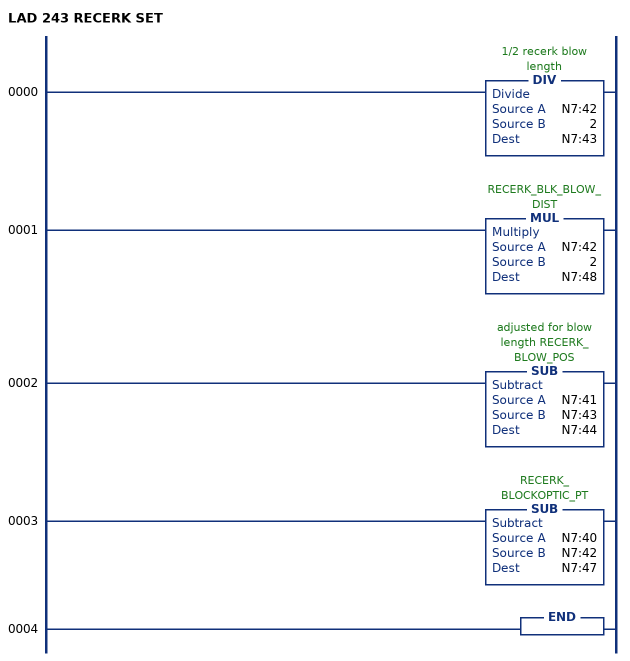
% Rung: 0 %
SOR DIV N7:42 2 N7:43 EOR
%   N7:42  RECERK_BLOW_LENGTH %
%   N7:43  "1/2 recerk blow length" %
% Rung: 1 %
SOR MUL N7:42 2 N7:48 EOR
%   N7:42  RECERK_BLOW_LENGTH %
%   N7:48  RECERK_BLK_BLOW_DIST %
% Rung: 2 %
SOR SUB N7:41 N7:43 N7:44 EOR
%   N7:41  RECERK_BLOW_POS_HMI  "recerk blow position set from hmi" %
%   N7:43  "1/2 recerk blow length" %
%   N7:44  RECERK_BLOW_POS  "adjusted for blow length" %
% Rung: 3 %
SOR SUB N7:40 N7:42 N7:47 EOR
%   N7:40  RECERK_OPTIC_POS %
%   N7:42  RECERK_BLOW_LENGTH %
%   N7:47  RECERK_BLOCKOPTIC_PT %
% Rung: 4 %
SOR END EOR

LADDER 244
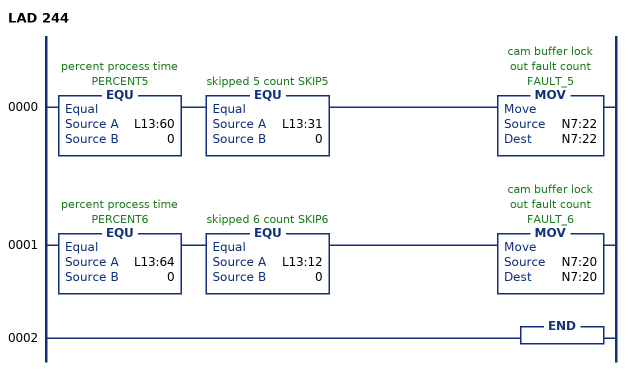
% Rung: 0 %
SOR EQU L13:60 0 EQU L13:31 0 MOV N7:22 N7:22 EOR
%   L13:60  PERCENT5  "percent process time" %
%   L13:31  SKIP5  "skipped 5 count" %
%   N7:22  FAULT_5  "cam buffer lock out fault count" %
% Rung: 1 %
SOR EQU L13:64 0 EQU L13:12 0 MOV N7:20 N7:20 EOR
%   L13:64  PERCENT6  "percent process time" %
%   L13:12  SKIP6  "skipped 6 count" %
%   N7:20  FAULT_6  "cam buffer lock out fault count" %
% Rung: 2 %
SOR END EOR

LADDER 249 "TESTOPTIC"
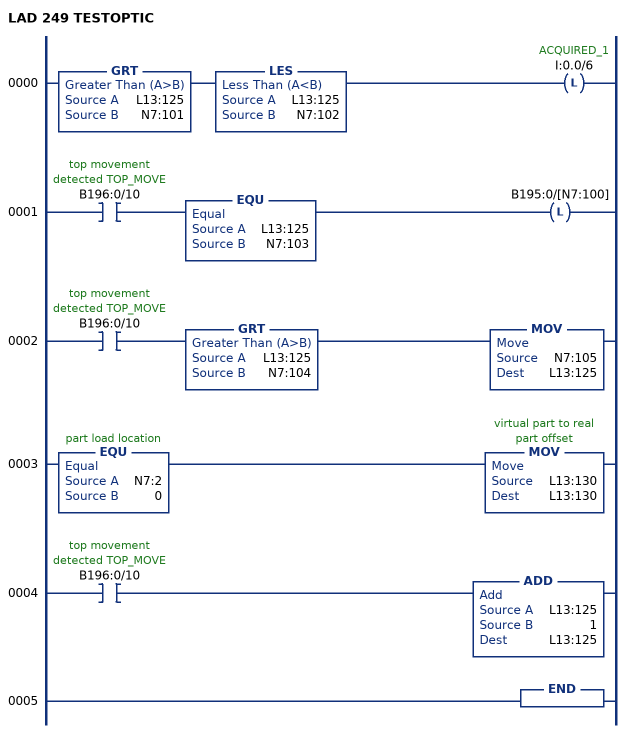
% Rung: 0 %
SOR GRT L13:125 N7:101 LES L13:125 N7:102 OTL I:0.0/6 EOR
%   I:0.0/6  ACQUIRED_1 %
% Rung: 1 %
SOR XIC B196:0/10 EQU L13:125 N7:103 OTL B195:0/[N7:100] EOR
%   B196:0/10  TOP_MOVE  "top movement detected" %
% Rung: 2 %
SOR XIC B196:0/10 GRT L13:125 N7:104 MOV N7:105 L13:125 EOR
%   B196:0/10  TOP_MOVE  "top movement detected" %
% Rung: 3 %
SOR EQU N7:2 0 MOV L13:130 L13:130 EOR
%   N7:2  "part load location" %
%   L13:130  "virtual part to real part offset" %
% Rung: 4 %
SOR XIC B196:0/10 ADD L13:125 1 L13:125 EOR
%   B196:0/10  TOP_MOVE  "top movement detected" %
% Rung: 5 %
SOR END EOR

LADDER 250 "RATE1"
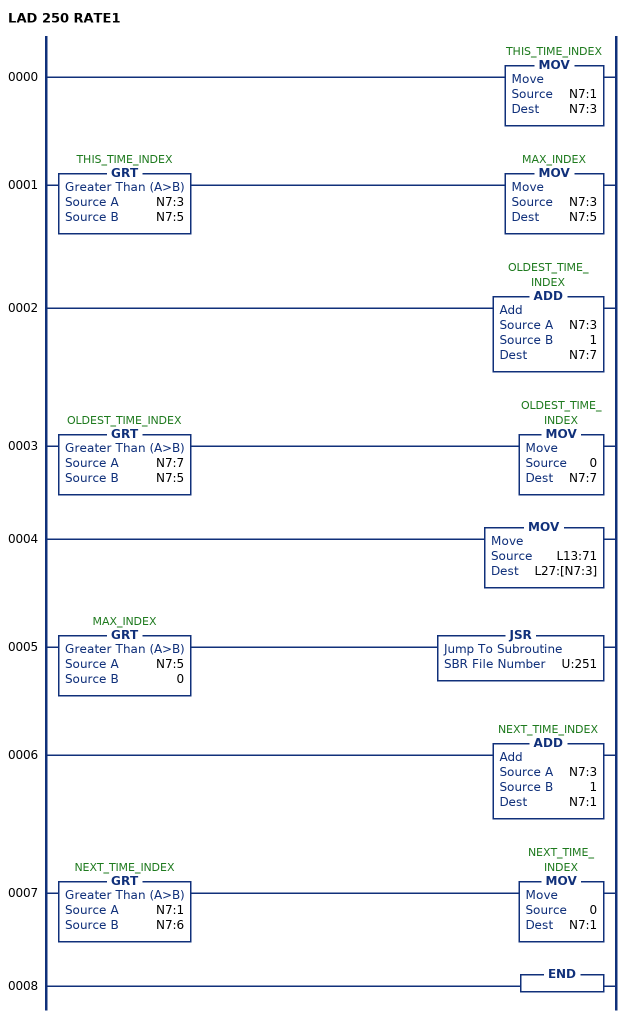
% Rung: 0 %
SOR MOV N7:1 N7:3 EOR
%   N7:1  NEXT_TIME_INDEX %
%   N7:3  THIS_TIME_INDEX %
% Rung: 1 %
SOR GRT N7:3 N7:5 MOV N7:3 N7:5 EOR
%   N7:3  THIS_TIME_INDEX %
%   N7:5  MAX_INDEX %
% Rung: 2 %
SOR ADD N7:3 1 N7:7 EOR
%   N7:3  THIS_TIME_INDEX %
%   N7:7  OLDEST_TIME_INDEX %
% Rung: 3 %
SOR GRT N7:7 N7:5 MOV 0 N7:7 EOR
%   N7:7  OLDEST_TIME_INDEX %
%   N7:5  MAX_INDEX %
% Rung: 4 %
SOR MOV L13:71 L27:[N7:3] EOR
%   L13:71  HSC_TIME %
%   N7:3  THIS_TIME_INDEX %
% Rung: 5 %
SOR GRT N7:5 0 JSR U:251 EOR
%   N7:5  MAX_INDEX %
% Rung: 6 %
SOR ADD N7:3 1 N7:1 EOR
%   N7:3  THIS_TIME_INDEX %
%   N7:1  NEXT_TIME_INDEX %
% Rung: 7 %
SOR GRT N7:1 N7:6 MOV 0 N7:1 EOR
%   N7:1  NEXT_TIME_INDEX %
%   N7:6  UPPER_INDEX_LIMIT  "buffer count 1" %
% Rung: 8 %
SOR END EOR

LADDER 251 "RATE2"
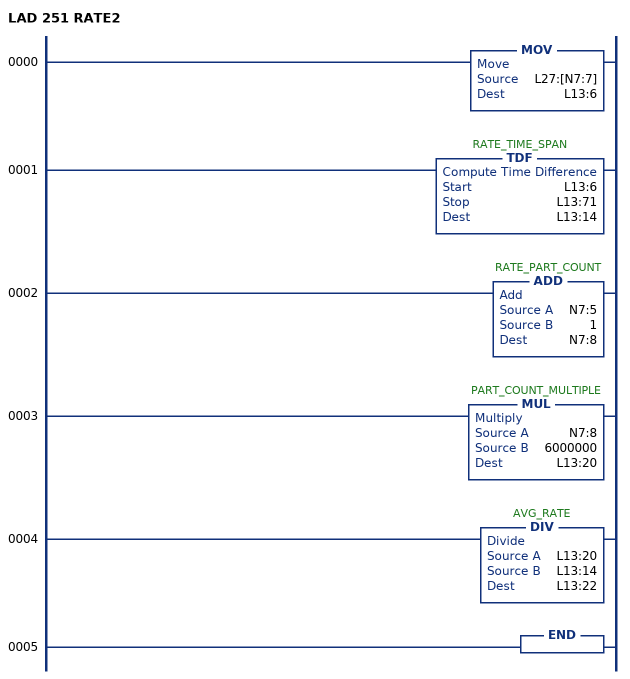
% Rung: 0 %
SOR MOV L27:[N7:7] L13:6 EOR
%   N7:7  OLDEST_TIME_INDEX %
% Rung: 1 %
SOR TDF L13:6 L13:71 L13:14 EOR
%   L13:71  HSC_TIME %
%   L13:14  RATE_TIME_SPAN %
% Rung: 2 %
SOR ADD N7:5 1 N7:8 EOR
%   N7:5  MAX_INDEX %
%   N7:8  RATE_PART_COUNT %
% Rung: 3 %
SOR MUL N7:8 6000000 L13:20 EOR
%   N7:8  RATE_PART_COUNT %
%   L13:20  PART_COUNT_MULTIPLE %
% Rung: 4 %
SOR DIV L13:20 L13:14 L13:22 EOR
%   L13:20  PART_COUNT_MULTIPLE %
%   L13:14  RATE_TIME_SPAN %
%   L13:22  AVG_RATE %
% Rung: 5 %
SOR END EOR

LADDER 252 "RESET RATE"
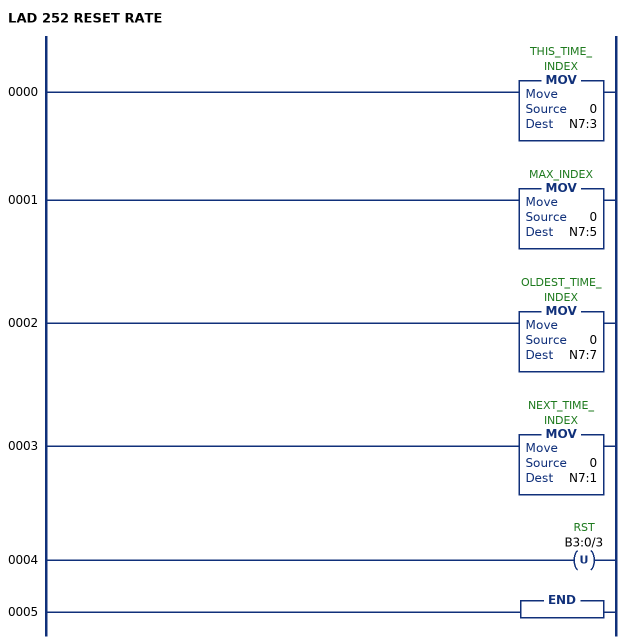
% Rung: 0 %
SOR MOV 0 N7:3 EOR
%   N7:3  THIS_TIME_INDEX %
% Rung: 1 %
SOR MOV 0 N7:5 EOR
%   N7:5  MAX_INDEX %
% Rung: 2 %
SOR MOV 0 N7:7 EOR
%   N7:7  OLDEST_TIME_INDEX %
% Rung: 3 %
SOR MOV 0 N7:1 EOR
%   N7:1  NEXT_TIME_INDEX %
% Rung: 4 %
SOR OTU B3:0/3 EOR
%   B3:0/3  RST %
% Rung: 5 %
SOR END EOR

LADDER 253 "UNUSED"
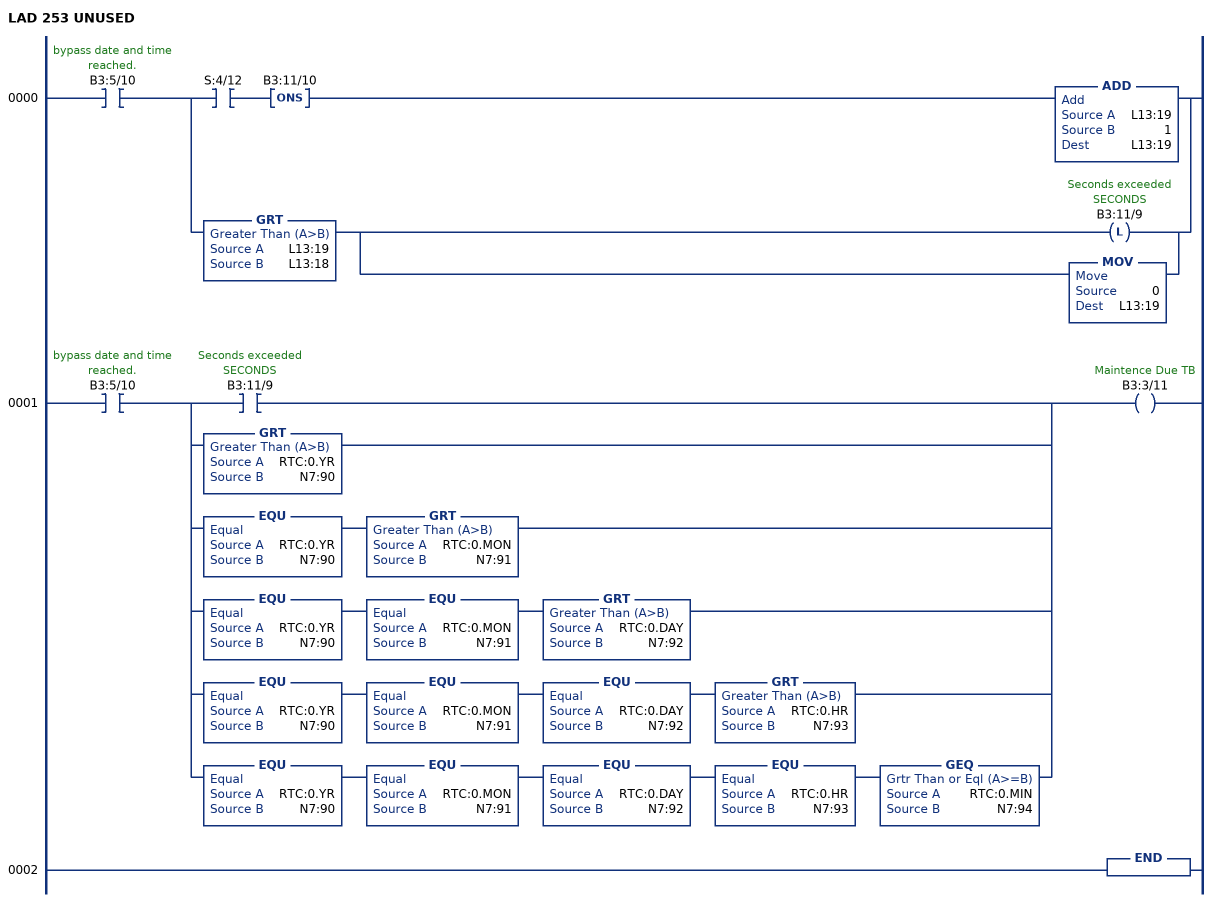
% Rung: 0 %
SOR XIC B3:5/10 BST XIC S:4/12 ONS B3:11/10 ADD L13:19 1 L13:19 NXB GRT L13:19 L13:18 BST OTL B3:11/9 NXB MOV 0 L13:19 BND BND EOR
%   B3:5/10  "bypass date and time reached." %
%   L13:18  MAX %
%   B3:11/9  SECONDS  "Seconds exceeded" %
% Rung: 1 %
SOR XIC B3:5/10 BST XIC B3:11/9 NXB GRT RTC:0.YR N7:90 NXB EQU RTC:0.YR N7:90 GRT RTC:0.MON N7:91 NXB EQU RTC:0.YR N7:90 EQU RTC:0.MON N7:91 GRT RTC:0.DAY N7:92 NXB EQU RTC:0.YR N7:90 EQU RTC:0.MON N7:91 EQU RTC:0.DAY N7:92 GRT RTC:0.HR N7:93 NXB EQU RTC:0.YR N7:90 EQU RTC:0.MON N7:91 EQU RTC:0.DAY N7:92 EQU RTC:0.HR N7:93 GEQ RTC:0.MIN N7:94 BND OTE B3:3/11 EOR
%   B3:5/10  "bypass date and time reached." %
%   B3:11/9  SECONDS  "Seconds exceeded" %
%   N7:90  RTC %
%   B3:3/11  TB  "Maintence Due" %
% Rung: 2 %
SOR END EOR

OTHER DOCUMENTED ADDRESSES
  I:0.0/0  TOP_CONV_ENC_A
  I:0.0/1  TOP_CONV_ENC_B
  PFILE:6  "check for part jams"
  PFILE:10  "Bottom belt HSC"
  PFILE:12  "Top belt HSC"
  Q2:55  END_OF_MAIN

COMMENTS NOT ATTACHED TO A CURRENT RUNG
  F8:13: *************************
    Loads Side Camera Passing data into a bit shift
    *************************
    
    loads passing data bit into passing data bit shift register at the part present cl.
  I:0.0/8: special rung for testing. This rung can simulate a pass signal. It will not be timed correctly.
  B23:0/0: Yet another bit shift load with data in the part position indicating that there was a bottom system part pass as well as a top system part present at this location.
    
    verified works w/bypassed 071910 and unbypassed 072010
  C5:4: tempory counting to verify pass part count with boxing part count.
  B22:0/0: ***********************
     Bottom Part Syncronizing Logic
    ***********************
    
    This is the point at the bottom of the top conveyor where the part jumps from the bottom conveyor.  This system will then track the part through the top system to the point of the laser optic in order to verify that the part in question has passed the bottom inspection.  I believe that we NEED to include FAILING inspections to eliminate the possibility of a out of position part from passing. LW 072010
  T20:2.ACC: This rung is starting a timer that should be activated directly before the laser optic part presense sensor on the top conveyer and should cause the top optic to be ignored if the bottom camera system didn't pass. however other arrangements must be made if the bottom camera isn't going to be used as is the case with a nut inspection.
  T20:2: The timer used to verify that the part that triggered the top laser optic has passed the bottom camer. needs to be count
  N17:8: ****************************************************************************************************************
    I can not find anywhere in the program where the "Test Spacing From Pickup to Trigger is activated indicating to me that this entire function must not be doing anything in this program at this time.
    ****************************************************************************************************************
  B11:0/0: load part present bit shit with one shot data from the part present sensor
  B3:7/9: ************************************
     The next 3 rungs appear to do nothing
    ***********************************
  B3:6/0: make a bit come on indicating that a part that passed the bottom camera is within  range when crossing the top camera.
  B3:6/1: ***********************
    Part Width and  Location
    ***********************
    
    Calculates the position of parts on the top belt by measureing the part width by calculating the number of belt movement pulses that occure when the optic is blocked and then devides that in half and add that to the optic location in the part presnet bit shift when the top optic is cleared.
  B9:0/[N7:47]: Remove any part present signals outside of expected location
  B9:0/[N7:50]: Remove any part present signals outside of expected location
  F19:0: Counter inside of a high speed counter interrupt counts the number of Bit Shifts that need to be processed in order to move the logic with the parts on the conveyor.
  F8:14: **************
    Bottom Top Camera Trigger
    *************
    
    Trigger Bottom Top Camera
  L13:104: Tracking error handler
  N10:4: test if boxing is connected
  B3:11/3: After initial delay allow blow two start functioning
  RUNG000150-000011: trigger count
  RUNG000150-000012: wipe stored part data if acq time expires
  RUNG000150-000013: clear data for aquire time expired
  RUNG000150-000014: clear data for time
  RUNG000150-000016: wiped count
  RUNG000150-000018: pass, fail and acquire inputs
  RUNG000150-000025: pass code / Set pass bit in Bit Shift
    captures result position and processing time
    Unlatch pass bit
  RUNG000150-000032: pass count
  RUNG000150-000035: fail count
  RUNG000150-000038: acquire code
  RUNG000150-000039: Grab trigger/acquire position
    Grab acquire time
  RUNG000150-000041: transfer tracked part positon from trigger/acquire to the acquire/result
    capture acquire time
    reset process time
  L13:101: record the minimum time between triggers
  L14:8: on when ok for run
  L14:3: off when ok to run
  L14:2: off when ok to run
  L14:5: on when ok to run, rear off turns both off
  L13:165: maximum q i1
  N7:76: removed relieance on trigger signal
  N197:20/0: Passes deformed head blowoff command to TOP PLC where solenoid output is located.
  L13:162: maximum q
  L13:163: maximum average q
  B3:10/1: prevents momentary signals from box present sensor from tripping the logic for box not present
    
    This is in responce to a problem created by the sensor occasionally turning on as if no box was in its path when there is a box present.
  B3:6/2: IF PROCESSING FAULT OCURES AT COUNTER SENSOR; CLEAR THE BELT OF PASSING DATA
  L14:23: ****************  nEEDS fIXING  **********************
  L14:36: ****************  nEEDS fIXING  **********************
  RUNG000010-000014: ****
                      Zeros out the non passing part count when one passes
    ****
  RUNG000010-000018: Remove any part present signals outside of expected location
  T4:27: Check for buffer reset
  T4:26: Check for buffer reset
  RUNG000125-000014: clear data for time
  RUNG000125-000013: clear data for aquire time expired
  RUNG000125-000012: wipe stored part data if acq time expires
  RUNG000125-000011: trigger count
  RUNG000125-000029: Set pass bit in Bit Shift
    captures result position and processing time
    Unlatch pass bit
  RUNG000125-000027: transfer tracked part positon from trigger/acquire to the acquire/result
    capture acquire time
    reset process time
  RUNG000125-000026: Grab trigger/acquire position
    Grab acquire time
  RUNG000125-000025: pass code / Set pass bit in Bit Shift
    captures result position and processing time
    Unlatch pass bit
  RUNG000125-000018: pass, fail and acquire inputs
  RUNG000125-000016: wiped count

REVISION NOTES
  13: updated count reset
  14: added io moduals
  15: multiple steps toward new hmi integration
  21: test

DATA TABLE (non-zero values as saved)
DATA B3
% B3:0 % 0X2000 0X0000 0X62C4 0XA408 0X0D26 0X0060 0X4000 0X0021 0X4007 0X0000
% B3:10 % 0X2041 0X0846 0X2000 0X0000
DATA T4
% .PRE .ACC %
% T4:0 % 300 0
% T4:1 % 150 151
% T4:2 % 600 0
% T4:3 % 32765 0
% T4:4 % 32765 0
% T4:5 % 666 0
% T4:6 % 10 32766
% T4:7 % 150 150
% T4:8 % 250 0
% T4:9 % 50 29
% T4:10 % 200 200
% T4:11 % 666 0
% T4:12 % 17 23
% T4:13 % 6 1
% T4:14 % 250 0
% T4:15 % 222 0
% T4:16 % 333 0
% T4:17 % 100 43
% T4:18 % 120 120
% T4:19 % 300 0
% T4:20 % 200 0
% T4:21 % 200 0
% T4:22 % 200 200
% T4:23 % 50 0
% T4:24 % 50 0
% T4:25 % 50 0
% T4:26 % 250 0
% T4:27 % 250 0
% T4:28 % 250 0
% T4:29 % 5000 0
% T4:30 % 50 50
% T4:31 % 20 0
% T4:32 % 69 0
DATA C5
% .PRE .ACC %
% C5:0 % 32766 0
DATA R6
% .LEN .POS %
% R6:0 % 2048 0
% R6:1 % 2048 0
% R6:2 % 3 0
% R6:3 % 3 0
% R6:4 % 1250 0
% R6:5 % 1250 0
% R6:6 % 1200 0
% R6:7 % 10 0
% R6:8 % 3 0
% R6:9 % 3 0
% R6:10 % 1440 0
% R6:11 % 928 0
% R6:12 % 10 0
% R6:13 % 10 0
% R6:14 % 10 0
% R6:15 % 10 0
% R6:16 % 1200 0
% R6:17 % 1440 0
% R6:18 % 928 0
% R6:19 % 10 0
DATA N7
% N7:0 % 666 0 1154 0 0 0 49 0 1 0
% N7:10 % 22 70 0 22 32767 250 777 666 250 94
% N7:20 % 1 93 20 0 0 34 34 32767 2 20
% N7:30 % 46 10 2 20 46 10 1503 333 1493 333
% N7:40 % 2020 2097 10 5 2092 10 21 2010 20 0
% N7:50 % 1236 0 175 16 0 0 0 1464 12 0
% N7:60 % 1 32767 4012 20 31 0 0 15 30 20
% N7:70 % 0 21 23 27738 32767 0 122 0 16 0
% N7:80 % 0 6 95 0 0 0 5 500 0 0
% N7:90 % 2011 4 4 12 1 0 0 0 0 1600
% N7:100 % 1003 90 110 100 175 25 0 0 0 0
DATA F8
% F8:0 % 18 206.64 23807 499 0.23807
% F8:5 % 0 0 500 1.9 2
% F8:10 % 1 0.08897486 0 101 63.26563
% F8:15 % 37.73437 4040 2 0 0
% F8:20 % 0 0.02 0 1 0
% F8:25 % 0 932781 0.222 279.6551 848597
% F8:30 % 0 170 0.03 38 852060
% F8:35 % 0 0 0 0 77
% F8:40 % 101 37.73437 0 100 1
% F8:45 % 1 2 0.21455 0 0
% F8:50 % 0 0 1 0 1
% F8:55 % 2000000 -221 0 0 0
% F8:95 % 0 0 0 492 4.92
DATA B9
% B9:130 % 0X0000 0X0000 0X0000 0X0000 0X2000 0X0000 0X0000 0X0000 0X0000 0X8000
% B9:140 % 0X2480 0X0000 0X0000 0X0000 0X0000 0X0000 0X0000 0X0000 0X0000 0X0000
% B9:160 % 0X0000 0X0000 0X0000 0X0000 0X0000 0X0000 0X2000 0X0002 0X0000 0X0000
% B9:170 % 0X0000 0X0000 0X0000 0X2000 0X0000 0X0000 0X0000 0X0000 0X0000 0X0000
% B9:180 % 0X0000 0X0000 0X0000 0X0000 0X0000 0X0002 0X0000 0X0000 0X0000 0X0000
% B9:190 % 0X0010 0X0000 0X0000 0X0000 0X0000 0X0000 0X0000 0X0000 0X0000 0X0000
% B9:200 % 0X2B64 0X2B64 0X0000 0X0010 0X0000 0X2000 0X0000 0X0000 0X0000 0X0000
% B9:220 % 0X0000 0X0000 0X0000 0X0200 0X0000 0X0000 0X0000 0X0000 0X0000 0X0020
% B9:230 % 0X0040 0X0000 0X0000 0X0000 0X0000 0X0000 0X0000 0X0000 0X0000 0X0000
DATA B11
% B11:180 % 0X0000 0X8000 0X0000 0X0000 0X0000 0X0000 0X0000 0X0000 0X0000 0X0000
% B11:240 % 0X0000 0X0000 0X0000 0X4000 0X0000 0X0000 0X0000 0X0000 0X0000 0X0000
DATA B12
% B12:0 % 0X0155 0X0000 0X0000 0X0000 0X0000 0X0000 0X0000 0X0000 0X0000 0X0000
DATA L13
% L13:0 % 308402300 308407124 4824 0 1000
% L13:5 % 1 1796853408 100 1162124017 1162124017
% L13:10 % 492 2147483647 0 0 1320294715
% L13:15 % 2073168201 -2147483648 2147483647 2147483647 82058
% L13:20 % 6000000 897100589 0 2000498310 884433458
% L13:25 % 25 0 72669925 0 777
% L13:30 % 2010317696 97 884450976 29 97
% L13:35 % 0 97 884450976 0 884433458
% L13:40 % 2010317725 0 61125062 20 0
% L13:45 % 60 700 70944452 12343079 12325561
% L13:50 % 83 20 444 20 444
% L13:55 % 0 0 62850570 225 336
% L13:60 % 9544372 3300 29 2147483647 6391320
% L13:65 % 0 20 -3 -1177857713 2002
% L13:70 % -1177813377 -1177813429 52 40 2000
% L13:75 % -2 0 109510 2000498335 1095
% L13:80 % 25 -20 150 200 200
% L13:85 % 16766 200 45 26483 1000
% L13:90 % 26616 0 0 1000 0
% L13:95 % 60 99000 99000 25989 99000
% L13:100 % -1478910248 1 2298 50 42
% L13:105 % 1 1 537010374 52 537010368
% L13:110 % 6 30 0 859995424 859995418
% L13:115 % 859995425 7 4 859995421 3
% L13:120 % 0 12018 0 30 49
% L13:125 % 164 19 155494060 137 155494060
% L13:130 % -3 1 -49 1 0
% L13:135 % 0 1000 111 12 0
% L13:140 % 0 11 12 0 20
% L13:145 % 2568 1273 1284 111 111
% L13:150 % -1538760531 -1538760111 88 0 100
% L13:155 % 420 332 24 0 37104441
% L13:160 % 3 18 4 395082 53203921
% L13:165 % 3 189116 95 13 8150
% L13:170 % 55946610 30 2868678 342419 0
% L13:175 % 0 0 45 32 38
% L13:180 % 176247033 25 99000 52866 644409
% L13:185 % 64 916459 92 627156 63
% L13:190 % 4 5 0 0 0
DATA F14
% F14:0 % 760.1599 200.1099 76 20 15
% F14:5 % 32766 21297.9 0 0 0
DATA N15
% N15:0 % 6 889 1924 1512 1502 134 98 1172 1150 10
% N15:10 % 61 504 0 0 0 0 1172 0 0 0
DATA L16
% L16:0 % 8 17 11 0 20
% L16:5 % 250 5000 5000 182 19
% L16:10 % 1256 18 2045 6599584 98
% L16:15 % 99 0 0 0 0
DATA B17
% B17:60 % 0XC000 0X0000 0X0000 0X0000 0X0000 0X0000 0X0000 0X0000 0X0000 0X0000
DATA B18
% B18:60 % 0XC000 0X0000 0X0000 0X0000 0X0000 0X0000 0X0000 0X0000 0X0000 0X0000
DATA L21
% L21:0 % 2010310030 2010310254 2010310479 2010310706 2010310931
% L21:5 % 2010311156 2010311381 2010311607 2010311834 2010312059
% L21:10 % 2010312285 2010312510 2010312735 2010312960 2010313186
% L21:15 % 2010313411 2010313636 2010313861 2010314087 2010314312
% L21:20 % 2010314538 2010314763 2010314988 2010315214 2010315441
% L21:25 % 2010315666 2010315892 2010316117 2010316342 2010316569
% L21:30 % 2010316795 2010317020 2010317246 2010317471 2010317696
% L21:35 % 2010306644 2010306870 2010307096 2010307321 2010307547
% L21:40 % 2010307772 2010307998 2010308224 2010308450 2010308676
% L21:45 % 2010308901 2010309127 2010309352 2010309578 2010309804
DATA L22
% L22:0 % 884449432 884449477 884449522 884449568 884449613
% L22:5 % 884449659 884449704 884449750 884449796 884449841
% L22:10 % 884449886 884449932 884449977 884450022 884450068
% L22:15 % 884450113 884450158 884450203 884450249 884450294
% L22:20 % 884450340 884450385 884450430 884450476 884450522
% L22:25 % 884450567 884450613 884450658 884450703 884450749
% L22:30 % 884450795 884450840 884450886 884450931 884450976
% L22:35 % 884448749 884448795 884448840 884448885 884448931
% L22:40 % 884448977 884449022 884449068 884449114 884449159
% L22:45 % 884449204 884449250 884449295 884449341 884449387
DATA L23
% L23:0 % 65535 -65536 -65536 -65536 -65536
% L23:5 % -65536 -65536 2 65535 -65536
% L23:10 % -65536 0 17 10 17
% L23:15 % 0 0 0 0 8
% L23:20 % 0 -65536 -65536 -65536 -65536
% L23:25 % -65536 20 19 20 0
% L23:30 % 0 0 -65536 -65536 -65536
% L23:35 % -65536 -65536 -65536 -65536 -65536
% L23:40 % 16270 18414 0 63266 -65536
% L23:45 % 5062 0 0 0 0
% L23:50 % 0 -65536 -65536 17 -65536
% L23:55 % 33 5079 -65536 0 0
% L23:60 % 0 -65536 -65536 -65536 0
DATA L24
% L24:0 % -65536 122 -65536 222 -65536
% L24:5 % 65535 -65536 -65536 -65536 -65536
% L24:10 % 50 27 0 1 23
% L24:15 % 1198 1030 95 18 30
% L24:20 % 30 -65536 1226 -65536 -65536
% L24:25 % 222 1236 -65536 -65536 222
% L24:30 % 1466 27 10000 -65536 55
% L24:35 % 180 -65536 180 65535 101
% L24:40 % 101 1000 -65536 -65536 10
% L24:45 % 222 192 -65536 0 -65536
% L24:50 % -999 30 10000 65535 900
DATA L25
% L25:0 % 2000490914 2000491251 2000491586 2000491923 2000492259
% L25:5 % 2000492596 2000492932 2000493269 2000493604 2000493940
% L25:10 % 2000494276 2000494612 2000494948 2000495285 2000495621
% L25:15 % 2000495957 2000496293 2000496630 2000496966 2000497301
% L25:20 % 2000497636 2000497974 2000498310 1997022512 1997022848
% L25:25 % 1997023184 1997023520 1997023856 1997024193 1997024529
% L25:30 % 1997024865 1997025202 1997025537 1997025874 1997026210
% L25:35 % 1997026546 1997026882 1997027217 1997027554 1997027890
% L25:40 % 1997028226 1997028562 2000488225 2000488562 2000488899
% L25:45 % 2000489235 2000489571 2000489908 2000490243 2000490579
DATA L26
% L26:0 % 884433458 884433458 884433458 884433458 884433458
% L26:5 % 884433458 884433458 884433458 884433458 884433458
% L26:10 % 884433458 884433458 884433458 884433458 884433458
% L26:15 % 884433458 884433458 884433458 884433458 884433458
% L26:20 % 884433458 884433458 884433458 884433458 884433458
% L26:25 % 884433458 884433458 884433458 884433458 884433458
% L26:30 % 884433458 884433458 884433458 884433458 884433458
% L26:35 % 884433458 884433458 884433458 884433458 884433458
% L26:40 % 884433458 884433458 884433458 884433458 884433458
% L26:45 % 884433458 884433458 884433458 884433458 884433458
DATA L27
% L27:0 % 1796853408 1796884254 1796957757 1797044744 1797061494
% L27:5 % 1797073276 1797104616 1797156934 1797178807 1797299369
% L27:10 % 1797410382 1797419826 1797426484 1797432733 1797548764
% L27:15 % 1797639679 1797654325 1797742322 1797748653 1797754308
% L27:20 % 1797768909 1798077280 1798162958 1798279083 1798401355
% L27:25 % 1798408310 1798472028 1799003759 1799195991 1799365744
% L27:30 % 1799510602 1799614126 1801153603 1796127821 1796140623
% L27:35 % 1796247376 1796259374 1796324189 1796332857 1796431745
% L27:40 % 1796439712 1796445777 1796513801 1796569851 1796575391
% L27:45 % 1796596583 1796639201 1796686981 1796694340 1796701097
DATA L42
% L42:0 % 41 0 0 0 0
% L42:5 % 45 45 45 0 0
% L42:20 % 0 0 32766 32766 0
% L42:50 % 0 30
DATA L183
% L183:0 % 1427522383 1427522384 1 1000000000 0
% L183:5 % 321 6 283 0 0
DATA N184
% N184:0 % 0 333 0 0 0 0 0 0 0 0
DATA B185
% B185:0 % 0X0200 0X0001 0X0000 0X0000 0X0000 0X0000 0X0000 0X0000 0X0000 0X0000
DATA N186
% N186:0 % 100 0 0 0 0 0 0 0 0 0
DATA L187
% L187:0 % 34 0 497 0 0
% L187:5 % 1063 0 0 0 0
DATA F188
% F188:0 % 6 66 11 44 29
DATA B189
% B189:0 % 0X00E0 0X0000 0X0000 0X0000 0X0000 0X0000 0X0000 0X0000 0X0000 0X0000
DATA L190
% L190:0 % 1 5 0 0 0
% L190:25 % 84 0 0 0 0
% L190:30 % 0 2 0 0 0
DATA B191
% B191:0 % 0X0000 0X0001 0X0000 0X0000 0X0000 0X0000 0X0000 0X0000 0X0000 0X0000
DATA L192
% L192:0 % -1444152502 266932201 5055 76 0
% L192:5 % 1000000 39200000 999 999 8
% L192:10 % 0 0 1 78 17
% L192:15 % -1177638709 332250347 860888 32 0
% L192:20 % 180 101000000 0 0 0
DATA F193
% F193:0 % 1.268652 0.315 0.022 6 760
% F193:5 % -0.8252563 0.2 -0.1650513 964.1756 31592.18
% F193:10 % 0.011 0.195 0.165 0.337 200
% F193:15 % 0.09407043 0.025 0.002351761 33.34737 1092.66
DATA B196
% B196:0 % 0X0034 0X9FF2 0X0001 0X0000 0X0000 0X0000 0X0000 0X0000 0X0000 0X0000
% B196:30 % 0XE800 0X9BFF 0XEBFF 0XFFDF 0XFFFF 0X0000 0X0000 0X0000 0X0000 0X0000
DATA N197
% N197:0 % 1560 150 500 2500 2500 14417 5555 300 150 0
% N197:10 % 4000 969 4 0 0 0 0 0 0 0
% N197:30 % 15 48 0 0 0 0 0 0 0 0
DATA B198
% B198:0 % 0X0009 0X0000 0X0000 0X0000 0X0000 0X0000 0X0000 0X0000 0X0000 0X0000
DATA L199
% L199:0 % 1 5571998 134 11 3579521
% L199:5 % 0 0 0 5 1267042
% L199:10 % 0 224 10256 556 0
% L199:15 % 0 0 0 278717848 518
% L199:20 % 28295 16430853 5001 5001 0
% L199:25 % 0 0 28329 1 3781224
% L199:30 % 21630086 251 3809367 15030467 111
% L199:35 % 555 555 0 0 0
DATA N200
% N200:0 % 2046 1231 985 2047 2045 1594 1241 2045 2045 2045
% N200:10 % 0 0 0 1277 178 2046 1000 2045 2045 1218
% N200:20 % 1555 0 0 0 0 0 0 0 0 0
% N200:30 % 0 0 32767 0 0 0 0 0 0 0
DATA L201
% L201:0 % 20 40 40 -3011735 44
% L201:5 % 96629277 0 0 -3010662 0
% L201:10 % 0 0 0 327 43
% L201:15 % 0 43 0 43 36830
DATA B202
% B202:0 % 0X2241 0X0000 0X0001 0X0000 0X0000 0X0000 0X0000 0X0000 0X0000 0X0000
DATA N203
% N203:0 % 115 115 116 333 334 333 444 0 445 444
% N203:10 % 555 556 555 0 0 0 0 0 0 0
DATA L204
% L204:0 % 333 333 333 1362 124
% L204:5 % 2000 2000 462 222 0
% L204:10 % 0 0 0 1327077052 1327077052
% L204:15 % 1327077052 1327077052 1 0 0
% L204:20 % 0 0 333 0 0
% L204:30 % 333 0 0 0 0
DATA F205
% F205:0 % 655.32 655.32 655.32 655.32 0
